TYPE ST_LSPM_States :
STRUCT
	eState			: E_LSPM_States; // State
	eLastState		: E_LSPM_States; // Last state
END_STRUCT
END_TYPE

(* stored: Version 1.1.0.1, ProductVersion 3.1.4024.4
   DUT ST_LSPM_States: Id {e35a4290-c042-4073-bdc1-734aeac97432} *)
